// TwinCAT 3 PLC project ProjectPLC
// ProgramVersion: 3.1.4024.0
// libraries:
//   Tc2_Standard, * (Beckhoff Automation GmbH)
//   Tc2_System, * (Beckhoff Automation GmbH)
//   Tc3_Module, * (Beckhoff Automation GmbH)
// project tree:
//   GVLs/ GVL_HMI.TcGVL
//   / PlcTask.TcTTO
//   POUs/FunctionBlocks/ FB_DrainValve.TcPOU, FB_Pump.TcPOU, FB_Tank.TcPOU
//   POUs/HMI/ HMI.TcPOU
//   POUs/ MAIN.TcPOU
//   POUs/Objects/ WaterTankFilling.TcPOU
// real-time tasks:
//   TASK PlcTask: cycle T#10ms, priority 20, ADS port 350
//   TASK PlcTask1: cycle T#10ms, priority 21, ADS port 351

CONFIGURATION ProjectPLC
    RESOURCE PLC ON TwinCAT3
        TASK PlcTask(INTERVAL := T#10ms, PRIORITY := 21);
        PROGRAM MAIN WITH PlcTask : MAIN;
    END_RESOURCE
END_CONFIGURATION

// ---- GVLs/GVL_HMI.TcGVL
{attribute 'qualified_only'}
VAR_GLOBAL
(*TANK*)
	rTankMaxCapacity				: REAL;
	rTankCurrentLevel				: REAL;
	bButtonResetSimilation			: BOOL;

(*PUMP*)
	bLampPumpIsOn					: BOOL;
	rPumpActualFlowRate				: REAL;
	rPumpNewFlowRate				: REAL;
	bButtonActualizePumpFlowRate	: BOOL;
	
(*DRAIN VALVE*)
	bLampDrainValveIsOn				: BOOL;
END_VAR

// ---- POUs/MAIN.TcPOU
PROGRAM MAIN
VAR
END_VAR

(*CALL POUs*)
	WaterTankFilling();
	HMI();

END_PROGRAM

// ---- POUs/Objects/WaterTankFilling.TcPOU
PROGRAM WaterTankFilling
VAR
	fbTank			: FB_Tank;
	fbPump			: FB_Pump;
	fbDrainValve	: FB_DrainValve;
END_VAR

(*EXECUTE FBs*)
	fbPump.Execute();
	fbDrainValve.Execute();
	
(*PUMP - UPDATE LEVEL UNTIL LEVEL HIGH*)
	IF fbPump.bIsOn THEN
		IF NOT fbTank.bLevelHigh THEN
			fbTank.UpdateLevel(
				rFlowRate 			:= fbPump.rFlowRate, 
				rTimeStepSec		:= TO_REAL(TO_LREAL(_TaskInfo[GETCURTASKINDEXEX()].CycleTime) / 10_000_000));
		ELSIF fbTank.bLevelHigh THEN
			fbPump.Stop();
		END_IF
	END_IF

(*DRAIN VALVE - UPDATE LEVEL UNTIL TANK EMPTY*)
	IF fbDrainValve.bIsOn THEN
		IF NOT fbTank.bIsEmpty THEN
			fbTank.UpdateLevel(
					rFlowRate 		:= fbDrainValve.rFlowRate,
					rTimeStepSec	:= TO_REAL(TO_LREAL(_TaskInfo[GETCURTASKINDEXEX()].CycleTime) / 10_000_000));
		ELSE
			fbDrainValve.Stop();
		END_IF
	END_IF

END_PROGRAM

// ---- POUs/FunctionBlocks/FB_Tank.TcPOU
FUNCTION_BLOCK FB_Tank
VAR_INPUT
END_VAR
VAR_OUTPUT
END_VAR
VAR
	_rCurrentLevel	: REAL;
	_rMaxCapacity	: REAL;	
	_bIsEmpty		: BOOL;

	bAlarmNextCycle	: BOOL;		//ADDITIONAL VARIABLE TO STOP PUMP BEFORE OVERFLOWING
END_VAR

PROPERTY bIsEmpty : BOOL
GET
//EMPTY WHEN CURRENT LEVEL IS 0
bIsEmpty	:= rCurrentLevel = 0.0;
END_GET
SET
END_SET
END_PROPERTY

PROPERTY bLevelHigh : BOOL
GET
//LEVEL IS HIGH IF CURRENT LEVEL IS EQUAL TO TANK MAX CAPACITY OR OVERFLOATING IN NEXT CYCLE
bLevelHigh	:= (rCurrentLevel = rMaxCapacity) OR bAlarmNextCycle;
END_GET
SET
END_SET
END_PROPERTY

PROPERTY bLevelLow : BOOL
GET
VAR
END_VAR
VAR CONSTANT
	LOW_LVL_TRESHOLD		: REAL := 1.0;		//LITER
END_VAR
bLevelLow	:= rCurrentLevel < LOW_LVL_TRESHOLD;
END_GET
SET
END_SET
END_PROPERTY

METHOD FB_init : BOOL
VAR_INPUT
	bInitRetains : BOOL; // if TRUE, the retain variables are initialized (warm start / cold start)
	bInCopyCode : BOOL;  // if TRUE, the instance afterwards gets moved into the copy code (online change)
END_VAR
//INITIALIZE TANK MAX CAPACITY
rMaxCapacity	:= 1000;
END_METHOD

PROPERTY rCurrentLevel : REAL
GET
rCurrentLevel	:= _rCurrentLevel;
END_GET
SET
_rCurrentLevel	:= rCurrentLevel;
END_SET
END_PROPERTY

METHOD Reset : BOOL
VAR_INPUT
END_VAR
//SET CURRENT TANK LEVEL TO 0
rCurrentLevel		:= 0.0;
END_METHOD

PROPERTY rMaxCapacity : REAL
GET
rMaxCapacity	:= _rMaxCapacity;
END_GET
SET
_rMaxCapacity	:= rMaxCapacity;
END_SET
END_PROPERTY

METHOD SetCapacity : BOOL
VAR_INPUT
	rCapacity		: REAL;
END_VAR
//SET CAPACITY
rMaxCapacity	:= rCapacity;
END_METHOD

METHOD UpdateLevel : BOOL
VAR_INPUT
	rFlowRate		: REAL;
	rTimeStepSec	: REAL;
END_VAR
VAR
	rCyclicLvlChange	: REAL;
END_VAR
(*1. CALCULATE NEW LEVEL*)
	rCyclicLvlChange	:= rFlowRate * rTimeStepSec;
	rCurrentLevel		:= rCurrentLevel + rCyclicLvlChange;

(*2. STOP IF OVERFLOWING IN NEXT CYCLE*)
	IF rCurrentLevel + rCyclicLvlChange > rMaxCapacity THEN
		bAlarmNextCycle		:= TRUE;
	ELSE
		bAlarmNextCycle		:= FALSE;
	END_IF
	
(*3. EMPTYING*)
	IF rCurrentLevel < 0 THEN
		Reset();
	END_IF
END_METHOD

END_FUNCTION_BLOCK

// ---- POUs/FunctionBlocks/FB_Pump.TcPOU
FUNCTION_BLOCK FB_Pump
VAR_INPUT
	bStartCmd	: BOOL;
	bStopCmd	: BOOL;
END_VAR
VAR_OUTPUT
END_VAR
VAR
	_bIsOn		: BOOL;
	_rFlowRate	: REAL;
END_VAR

PROPERTY bError : BOOL
GET
//ERROR STATE IF 'bStartCmd' IS ON AND PUMP IS NOT ON
bError	:= bStartCmd AND NOT bIsOn;
END_GET
SET
END_SET
END_PROPERTY

PROPERTY bIsOn : BOOL
GET
bIsOn	:= _bIsOn;
END_GET
SET
_bIsOn	:= bIsOn;
END_SET
END_PROPERTY

METHOD Execute : BOOL
VAR_INPUT
END_VAR
//CHECK ON STATE
IF bStartCmd THEN
	bIsOn		:= TRUE;
ELSIF bStopCmd THEN
	bIsOn		:= FALSE;
END_IF
END_METHOD

METHOD FB_init : BOOL
VAR_INPUT
	bInitRetains : BOOL; // if TRUE, the retain variables are initialized (warm start / cold start)
	bInCopyCode : BOOL;  // if TRUE, the instance afterwards gets moved into the copy code (online change)
END_VAR
//FLOW RATE NITIALIZATION
rFlowRate	:= 50.0;
END_METHOD

PROPERTY rFlowRate : REAL
GET
rFlowRate	:= _rFlowRate;
END_GET
SET
_rFlowRate	:= rFlowRate;
END_SET
END_PROPERTY

METHOD SetFlowRate : BOOL
VAR_INPUT
	rRate	: REAL;
END_VAR
//SET RATE
rFlowRate	:= rRate;
END_METHOD

ACTION Stop:
//SET COMMANDS TO STOP
bStartCmd	:= FALSE;
bStopCmd	:= TRUE;
END_ACTION

END_FUNCTION_BLOCK

// ---- POUs/FunctionBlocks/FB_DrainValve.TcPOU
FUNCTION_BLOCK FB_DrainValve EXTENDS FB_Pump
VAR_INPUT
END_VAR
VAR_OUTPUT
END_VAR
VAR
END_VAR

METHOD FB_init : BOOL
VAR_INPUT
	bInitRetains : BOOL; // if TRUE, the retain variables are initialized (warm start / cold start)
	bInCopyCode : BOOL;  // if TRUE, the instance afterwards gets moved into the copy code (online change)
END_VAR
//FLOW RATE NITIALIZATION
rFlowRate	:= -30.0;
END_METHOD

END_FUNCTION_BLOCK

// ---- POUs/HMI/HMI.TcPOU
PROGRAM HMI
VAR
END_VAR

(*RESET SIMULATION*)
	IF GVL_HMI.bButtonResetSimilation THEN
		WaterTankFilling.fbTank.Reset();
		GVL_HMI.bButtonResetSimilation	:= FALSE;
	END_IF

(*TANK*)
	GVL_HMI.rTankMaxCapacity	:= WaterTankFilling.fbTank.rMaxCapacity;
	GVL_HMI.rTankCurrentLevel	:= WaterTankFilling.fbTank.rCurrentLevel;

(*LAMPS*)
	GVL_HMI.bLampPumpIsOn		:= WaterTankFilling.fbPump.bIsOn;
	GVL_HMI.bLampDrainValveIsOn	:= WaterTankFilling.fbDrainValve.bIsOn;
	
(*PUMP FLOW RATE*)
	GVL_HMI.rPumpActualFlowRate	:= WaterTankFilling.fbPump.rFlowRate;
	
	IF GVL_HMI.bButtonActualizePumpFlowRate THEN
		WaterTankFilling.fbPump.SetFlowRate(rRate := GVL_HMI.rPumpNewFlowRate);
		GVL_HMI.bButtonActualizePumpFlowRate	:= FALSE;
	END_IF

END_PROGRAM
